// TIA Portal project "Zanzeta_L01_190722" (V16)

(* hardware
DEVICE "S7-1200 station_1"  S7-1200 Station
   slot 0: "Rack_0"  S7-1200 Rack  Rack  V1.0
   slot 1: "PLC_1"  CPU 1215C DC/DC/Rly  6ES7 215-1HG40-0XB0  V4.4
*)

// ===== PLC "PLC_1"  CPU 1215C DC/DC/Rly =====

VAR_GLOBAL   // PLC tag table "Default tag table"
   "Tag_1" AT %MD100 : DInt;
   "Tag_2" AT %MW101 : Int;
   "Tag_3" AT %MD102 : Real;
   "Tag_4" AT %I0.0 : Bool;
   "Tag_5" AT %M0.0 : Bool;
   "Tag_6" AT %MW104 : Int;
   "Tag_7" AT %I0.7 : Bool;
   "Tag_8" AT %Q0.1 : Bool;
END_VAR

// folder: LBC

TYPE "LBC_typeDiagnostics"
TITLE = LBC_typeDiagnostic
// Module related diagnostic information
   STRUCT
      status : Word;   // 16#0000-16#7FFF: Status of the FB 16#8000-16#FFFF: Error identification
      subfunctionStatus : Word;   // Status or return value of called FB's, FCs, system blocks or other status information
      stateNumber : DInt;   // State in the state machine of the block where the error occurred
   END_STRUCT;
END_TYPE

TYPE "LBC_typeInterfaceCommands"
TITLE = LBC_typeInterfaceCommands
// Module related commands from external systems
   STRUCT
      refreshConfiguration : Bool;   // TRUE: Copy global configuration parameters into module interface for external systems
      editConfiguration : Bool;   // TRUE: Edit mode for configuration parameters in control system is active - copying into module interface is stopped
      saveConfiguration : Bool;   // TRUE: Save configuration parameters from module interface into to global configuration parameters after change
      acknowledge : Bool;   // TRUE: Module error acknowledge / reset of errors in function block
   END_STRUCT;
END_TYPE

// folder: LBC/AnalogSignals/Scale

TYPE "LBC_typeAnalogScaleInterface"
TITLE = LBC_typeAnalogScaleInterface
// Module interface for external systems
   STRUCT
      commands : "LBC_typeInterfaceCommands";
      configuration : "LBC_typeAnalogScaleConfiguration";
      monitoring : "LBC_typeAnalogScaleValues";
      diagnostics : "LBC_typeDiagnostics";
   END_STRUCT;
END_TYPE

TYPE "LBC_typeAnalogScaleValues"
TITLE = LBC_typeAnalogScaleValues
// Module related monitoring information
   STRUCT
      enable : Bool;   // TRUE: Enable functionality of FB
      simulation : Bool;   // TRUE: Enable simulation input of input value
      inputValue : LReal;   // Value to be converted
      outputValue : LReal;   // Processed and scaled value
      minValueReached : Bool;   // Minimum configured process value reached. Value is limited to the minimum configured value.
      maxValueReached : Bool;   // Maximum configured process value reached. Value is limited to the maximum configured value.
      error : Bool;   // TRUE: An error occurred while processing the FB
   END_STRUCT;
END_TYPE

TYPE "LBC_typeAnalogScaleConfiguration"
TITLE = LBC_typeAnalogScaleConfiguration
// Module related configuration parameters
   STRUCT
      referenceDesignator : String[20] := 'AnalogScale';   // Device name or device ID
      physicalUnitInput : String[10] := 'unit';   // Physical unit (like [°C], [kWh], etc.) for the input value
      physicalUnitOutput : String[10] := 'unit';   // Physical unit (like [°C], [kWh], etc.) for the output value
      default : LReal := 0.0;   // Default OUTPUT value to be returned if function block is not enabled or quality is bad
      inputValueMax : LReal := 100.0;   // Maximum limit of the process value
      inputValueMin : LReal := -100.0;   // Minimum limit of the process value
      scaleInputUppPoint : LReal := 100.0;   // Upper point for the process value
      scaleInputLowPoint : LReal := -100.0;   // Lower point for the process value
      scaleOutputUppPoint : LReal := 200.0;   // Upper point for the analog process output
      scaleOutputLowPoint : LReal := -200.0;   // Lower point for the analog process output
      disableAlarms : Bool;   // TRUE: Disable the alarms of the block
   END_STRUCT;
END_TYPE

// folder: (top level)

DATA_BLOCK "CMD_PROS_DB"   // DB1
{ S7_Optimized_Access := 'TRUE' }
VERSION : 0.1
// stored: InstanceOfName CMD_PROS
"CMD_PROS"
BEGIN
END_DATA_BLOCK

DATA_BLOCK "TemplateStateMachine_DB"   // DB5
{ S7_Optimized_Access := 'TRUE' }
VERSION : 0.1
// stored: InstanceOfName TemplateStateMachine
"TemplateStateMachine"
BEGIN
END_DATA_BLOCK

// folder: DB

DATA_BLOCK "GlobalDB"   // DB2
{ S7_Optimized_Access := 'TRUE' }
VERSION : 0.1
   VAR RETAIN
      outScale_1 : Real;
      outScale_2 : DInt;
   END_VAR
   VAR
      spMin_1 : Int := 0;
      spMax1 : Int := 27468;
      spMin_2 : Real := 0.0;
      spMax_2 : Real := 20.0;
   END_VAR
   VAR RETAIN
      State_Value : Byte := 2;
   END_VAR
BEGIN
END_DATA_BLOCK

DATA_BLOCK "DB1_IO"   // DB3
{ S7_Optimized_Access := 'TRUE' }
VERSION : 0.1
   VAR
      DBX : Array[0..16] of Bool;
      DBY : Array[0..16] of Bool;
   END_VAR
   VAR RETAIN
      AX1 : DInt;
      AY1 : DInt;
   END_VAR
BEGIN
   DBX[0] := true;
   DBX[1] := true;
END_DATA_BLOCK

DATA_BLOCK "Alarm_DB"   // DB4
{ S7_Optimized_Access := 'TRUE' }
VERSION : 0.1
   VAR
      Alarm_Bool : Array[0..15] of Bool;
   END_VAR
BEGIN
END_DATA_BLOCK

// folder: (top level)

FUNCTION_BLOCK "CMD_PROS"   // FB1, LAD
{ S7_Optimized_Access := 'TRUE' }
VERSION : 0.1
BEGIN
END_FUNCTION_BLOCK

FUNCTION_BLOCK "TemplateStateMachine"   // FB2, LAD
{ S7_Optimized_Access := 'TRUE' }
VERSION : 0.1
   VAR_INPUT
      Actual_Step : Byte;
      Desire_Step : Byte;
      Number_Step : Byte;
      Action_Condirion : Byte;
      Safety_Condition : Byte;
      Interlock : Bool;
      Transition_Condition : Bool;
      Exceptional_Transition : Bool;
      Value : Byte;
   END_VAR
   VAR_OUTPUT
      Actual_Step_1 : Byte;
      Action1 : Bool;
      Action2 : Bool;
      Action3 : Byte;
   END_VAR
   VAR_TEMP   // added for the SCL form of the ladder/FBD networks
      _w1 : Bool;
   END_VAR
BEGIN

REGION Network 1
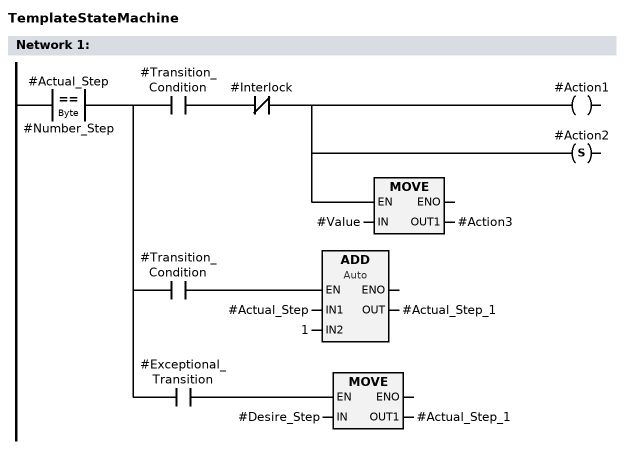
   RUNG wire#powerrail
      { S7_Templates := "SrcType := Byte" } EQ_Contact(in1 := #Actual_Step, in2 := #Number_Step)
      wire#w1
      Contact( #Transition_Condition )
      I_Contact( #Interlock )
      wire#w2
      Coil( #Action1 )
   END_RUNG
   RUNG wire#w2
      S_Coil( #Action2 )
   END_RUNG
   RUNG wire#w2
      Move(in := #Value, out1 => #Action3)
   END_RUNG
   RUNG wire#w1
      Contact( #Transition_Condition )
      Add(in1 := #Actual_Step, in2 := 1, out => #Actual_Step_1)
   END_RUNG
   RUNG wire#w1
      Contact( #Exceptional_Transition )
      Move(in := #Desire_Step, out1 => #Actual_Step_1)
   END_RUNG
   // the same network as SCL:
   #_w1 := #Actual_Step = #Number_Step;
   #Action1 := #_w1 AND #Transition_Condition AND NOT #Interlock;
   IF #Action1 THEN
       #Action2 := TRUE;
       #Action3 := #Value;
   END_IF;
   IF #_w1 AND #Transition_Condition THEN #Actual_Step_1 := #Actual_Step + 1; END_IF;
   IF #_w1 AND #Exceptional_Transition THEN #Actual_Step_1 := #Desire_Step; END_IF;
END_REGION
END_FUNCTION_BLOCK

FUNCTION_BLOCK "LBC_AnalogScale"   // FB22004, SCL
TITLE = LBC_AnalogScale
{ S7_Optimized_Access := 'TRUE' }
AUTHOR : Siemens_Digital_Industry
FAMILY : LBC
NAME : LBC_AnalogScale
// The function is used for processing (scaling) an analog process value to another process value of a different range.  
// Converts it from one to another meaningful unit, e.g. $[rpm]$ to $[m/s]$, $[°C]$ to $[°F]$.
   VAR_INPUT
      enable : Bool;   // TRUE: Enable functionality of FB
      inputValue : LReal;   // Value to be converted
      simulation : Bool;   // TRUE: Enable simulation (input value)
      simulatedInputValue : LReal;   // Simulated input value
   END_VAR
   VAR_OUTPUT
      error : Bool;   // FALSE: No error TRUE: An error occurred during the execution of the FB
      status : Word := 16#7000;   // 16#0000-16#7FFF: Status of the FB 16#8000-16#FFFF: Error identification (see following Table)
      outputValue : LReal;   // Processed and scaled value
      maxValueReached : Bool;   // Maximum configured process value reached. Value is limited to the maximum configured value.
      minValueReached : Bool;   // Minimum configured process value reached. Value is limited to the minimum configured value.
   END_VAR
   VAR_IN_OUT
      configuration : "LBC_typeAnalogScaleConfiguration";
      moduleInterface : "LBC_typeAnalogScaleInterface";
   END_VAR
   VAR
      statProcessValues : "LBC_typeAnalogScaleValues";
      statDiagnostics : "LBC_typeDiagnostics";
      statReferenceDesignator : String[20];   // Device name or device ID
      statLimitationMessage : String[40];   // String to collect information for alarm message of value limitation
      statDisableAlarms : Bool;   // TRUE: Disable the alarms of the block
      statEnablePrevious : Bool;   // Previous value of 'enable' input
   END_VAR
   VAR CONSTANT
      STATUS_NO_ERROR_OCCURRED : Word := 16#0000;   // Status: No error occurred during execution
      STATUS_NO_CALL : Word := 16#7000;   // Status: Function block is not enabled
      STATUS_ENABLED : Word := 16#7002;   // Status: Function block is enabled
      ERR_RANGE_PARAMETRIZATION : Word := 16#8201;   // Error: Configuration range of parameters. min >= max
      ERR_SCALE_ANALOG_POINTS : Word := 16#8202;   // Error: Configuration of analog input points. Process Lower >= Upper
   END_VAR
   // statDiagnostics.status := 16#7000;
BEGIN
   REGION BLOCK INFO HEADER
     //===============================================================================
     // Siemens AG / (c)Copyright 2020
     //-------------------------------------------------------------------------------
     // Title:            LBC_AnalogScale
     // Comment/Function: The function is used for processing (scaling) an analog process value to another process value of a different range. 
     //                   Converts it from one to another meaningful unit, e.g. $[rpm]$ to $[m/s]$, $[°C]$ to $[°F]$.
     // Library/Family:   LBC - Library of Basic Control modules
     // Author:           Siemens Digital Industries
     // Tested with:      S7-PLCSIM Advanced 3.0
     // Engineering:      TIA Portal V16
     // Restrictions:     ENO mechanism is not used - forced to true.
     // Requirements:     PLC (S7-1200 / S7-1500)
     //-------------------------------------------------------------------------------
     // Change log table:
     // Version  | Date       | Expert in charge        | Changes applied
     //----------|------------|-------------------------|-----------------------------
     // 01.00.00 | 15.02.2021 | SIMATIC Systems Support | First released version
     //===============================================================================
   END_REGION

   REGION DESCRIPTION
   (/*The analog scale function block converts a process value to another process value of a different range, e.g. $[rpm]$ to $[m/s]$, $[°C]$ to $[°F]$.

   The processing of the function is started by assigning `TRUE` signal to the `enable` input.  
   If the block is enabled (logical `TRUE`) then the output value is scaled according to settings of the block.

   In order to ensure, that scaling works correctly, it is necessary to set the minimum and the maximum values for input and output.

   For further information see the explanation in the picture and math formulas below.

   ## Process chart
   ![LBC_AnalogScale](LBC_AnalogScale.png "LBC_AnalogScale")

   $ dx = x2 - x1 = scaleInputUppPoint - scaleInputLowPoint $  
   $ dy = y2 - y1 = scaleOutputUppPoint - scaleOutputLowPoint $

   ### Math equation
   $ y = \frac{y_2 - y_1}{x_2 - x_1} \cdot (x - x_1) + y_1 $

   $ x = inputValue $  
   $ y = outputValue $  
   $ x_1 = scaleInputLowPoint $  
   $ x_2 = scaleInputUppPoint $  
   $ y_1 = scaleOutputLowPoint $  
   $ y_2 = scaleOutputUppPoint $*/)
   END_REGION DESCRIPTION

   REGION PROCESS INPUT SIGNALS
     // Assign and initialize internal variables
     #statProcessValues.enable := #enable;
     #statProcessValues.simulation := #simulation;

     // Check if simulation is activated
     IF #statProcessValues.simulation THEN
       #statProcessValues.inputValue := #simulatedInputValue;
     ELSE
       #statProcessValues.inputValue := #inputValue;
     END_IF;

     // Reset limit bits
     #statProcessValues.maxValueReached := FALSE;
     #statProcessValues.minValueReached := FALSE;

     // Copy configuration to static for usage in supervision
     #statDisableAlarms := #configuration.disableAlarms;
   END_REGION PROCESS INPUT SIGNALS

   REGION PARAMETER CHECK
     // Check parameter if block is enabled
     IF #statProcessValues.enable THEN
       #statDiagnostics.status := #STATUS_ENABLED;
       // Validation for hardware range limits 
       // Check if parameters for hardware signal limits are within correct values
       IF #configuration.inputValueMin >= #configuration.inputValueMax THEN
         #statProcessValues.outputValue := #configuration.default;
         #statDiagnostics.status := #ERR_RANGE_PARAMETRIZATION;

       ELSIF #configuration.scaleInputLowPoint >= #configuration.scaleInputUppPoint THEN
         #statProcessValues.outputValue := #configuration.default;
         #statDiagnostics.status := #ERR_SCALE_ANALOG_POINTS;
       END_IF;
     END_IF;
   END_REGION PARAMETER CHECK

   REGION ENABLING/DISABLING
     IF #enable AND NOT #statEnablePrevious THEN
       // Copy configuration to static for usage in associated value of supervision
       #statReferenceDesignator := #configuration.referenceDesignator;

       // Initializes moduleInterface configuration with process configuration
       #moduleInterface.configuration := #configuration;
     END_IF;
     #statEnablePrevious := #enable;
   END_REGION ENABLING/DISABLING

   REGION PROCESS LOGIC
     // Use default value and set no call status if block is disabled
     IF NOT #statProcessValues.enable THEN
       #statProcessValues.outputValue := #configuration.default;
       #statDiagnostics.status := #STATUS_NO_CALL;

       // In case of Error return default
     ELSIF #statDiagnostics.status.%X15 THEN
       #statProcessValues.outputValue := #configuration.default;

       // No error - do process
     ELSE
       // Write status message, set no error
       #statDiagnostics.status := #STATUS_NO_ERROR_OCCURRED;

       // Check if process values are within the configured range
       IF #statProcessValues.inputValue < #configuration.inputValueMin THEN
         #statProcessValues.inputValue := #configuration.inputValueMin;
         #statProcessValues.minValueReached := TRUE;
         #statLimitationMessage := CONCAT(IN1 := LREAL_TO_STRING(#statProcessValues.inputValue), IN2 := #configuration.physicalUnitInput, IN3 := ' <= ', IN4 := LREAL_TO_STRING(#configuration.inputValueMin), IN5 := #configuration.physicalUnitOutput);

       ELSIF #statProcessValues.inputValue > #configuration.inputValueMax THEN
         #statProcessValues.inputValue := #configuration.inputValueMax;
         #statProcessValues.maxValueReached := TRUE;
         #statLimitationMessage := CONCAT(IN1 := LREAL_TO_STRING(#statProcessValues.inputValue), IN2 := #configuration.physicalUnitInput, IN3 := ' >= ', IN4 := LREAL_TO_STRING(#configuration.inputValueMax), IN5 := #configuration.physicalUnitOutput);

       ELSE // Clear alarm message string
         #statLimitationMessage := '';
       END_IF;

       // Scaling the process input
       #statProcessValues.outputValue := (((#statProcessValues.inputValue - #configuration.scaleInputLowPoint) / (#configuration.scaleInputUppPoint - #configuration.scaleInputLowPoint))
       * (#configuration.scaleOutputUppPoint - #configuration.scaleOutputLowPoint) + #configuration.scaleOutputLowPoint);

     END_IF;
   END_REGION PROCESS LOGIC

   REGION CONFIGURATION HANDLING
     // Refresh module interface configuration with process configuration
     IF #moduleInterface.commands.refreshConfiguration AND NOT #moduleInterface.commands.editConfiguration THEN
       #moduleInterface.configuration := #configuration;
     END_IF;
     #moduleInterface.commands.refreshConfiguration := FALSE;

     // Save module interface configuration to process configuration
     IF #moduleInterface.commands.saveConfiguration AND #moduleInterface.commands.editConfiguration THEN
       #configuration := #moduleInterface.configuration;
       #statReferenceDesignator := #configuration.referenceDesignator;
       #moduleInterface.commands.saveConfiguration := FALSE;
     END_IF;
   END_REGION CONFIGURATION HANDLING

   REGION PROCESS OUTPUT SIGNALS
     REGION Write Process data to module interface
       #statProcessValues.error := #statDiagnostics.status.%X15;
       #moduleInterface.monitoring := #statProcessValues;
       #moduleInterface.diagnostics := #statDiagnostics;
     END_REGION Write Process data to module interface

     REGION Write work data to interface and outputs    
       // Write application specific static values to outputs
       #outputValue := #statProcessValues.outputValue;
       #minValueReached := #statProcessValues.minValueReached;
       #maxValueReached := #statProcessValues.maxValueReached;

       // Function status
       #error := #statDiagnostics.status.%X15;
       #status := #statDiagnostics.status;
       // ENO mechanism disabled, ENO - forced to true
       ENO := TRUE;
     END_REGION Write static values to outputs
   END_REGION
END_FUNCTION_BLOCK

FUNCTION "Scalling" : Void   // FC1, LAD
{ S7_Optimized_Access := 'TRUE' }
VERSION : 0.1
   VAR_INPUT
      inMin1 : DInt;
      inMax1 : DInt;
      inMin2 : Real;
      inMax2 : Real;
      inValue : DInt;
   END_VAR
   VAR_OUTPUT
      outReal : LReal;
   END_VAR
   VAR_TEMP
      tempOutNorm1 : LReal;
   END_VAR
BEGIN

REGION Network 1
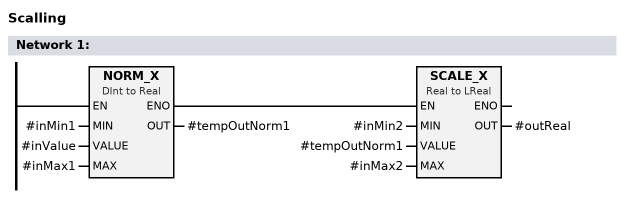
   RUNG wire#powerrail
      { S7_Templates := "[SrcType := DInt, DestType := Real]" } Normalize(min := #inMin1, value := #inValue, max := #inMax1, out => #tempOutNorm1)
      { S7_Templates := "[SrcType := Real, DestType := LReal]" } Scale(min := #inMin2, value := #tempOutNorm1, max := #inMax2, out => #outReal)
   END_RUNG
   // the same network as SCL:
   #tempOutNorm1 := NORM_X(MIN := #inMin1, VALUE := #inValue, MAX := #inMax1);
   #outReal := SCALE_X(MIN := #inMin2, VALUE := #tempOutNorm1, MAX := #inMax2);
END_REGION
END_FUNCTION

FUNCTION "RunMainMotor" : Void   // FC2, LAD
{ S7_Optimized_Access := 'TRUE' }
VERSION : 0.1
BEGIN

REGION Network 1
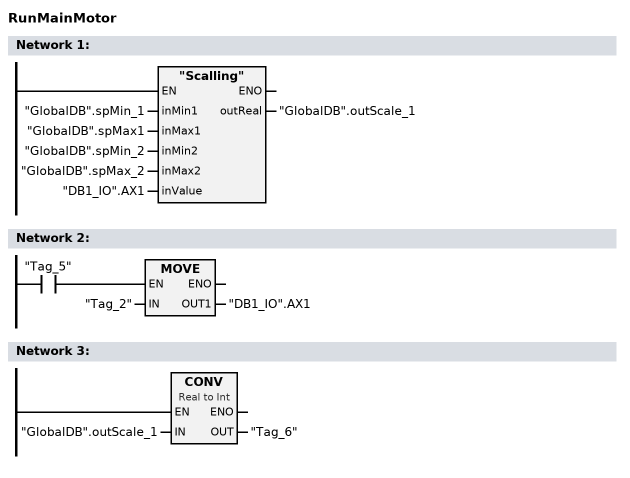
   RUNG wire#powerrail
      "Scalling"(inMin1 := "GlobalDB".spMin_1, inMax1 := "GlobalDB".spMax1, inMin2 := "GlobalDB".spMin_2, inMax2 := "GlobalDB".spMax_2, inValue := "DB1_IO".AX1, outReal => "GlobalDB".outScale_1)
   END_RUNG
   // the same network as SCL:
   "Scalling"(inMin1 := "GlobalDB".spMin_1,
              inMax1 := "GlobalDB".spMax1,
              inMin2 := "GlobalDB".spMin_2,
              inMax2 := "GlobalDB".spMax_2,
              inValue := "DB1_IO".AX1,
              outReal => "GlobalDB".outScale_1);
END_REGION

REGION Network 2
   RUNG wire#powerrail
      Contact( "Tag_5" )
      Move(in := "Tag_2", out1 => "DB1_IO".AX1)
   END_RUNG
   // the same network as SCL:
   IF "Tag_5" THEN "DB1_IO".AX1 := "Tag_2"; END_IF;
END_REGION

REGION Network 3
   RUNG wire#powerrail
      { S7_Templates := "[SrcType := Real, DestType := Int]" } Convert(in := "GlobalDB".outScale_1, out => "Tag_6")
   END_RUNG
   // the same network as SCL:
   "Tag_6" := REAL_TO_INT("GlobalDB".outScale_1);
END_REGION
END_FUNCTION

FUNCTION "IO_ASSIGMENT" : Void   // FC3, LAD
{ S7_Optimized_Access := 'TRUE' }
VERSION : 0.1
BEGIN

REGION Network 1 (SCL)
   REGION io
       // Statement section REGION

   END_REGION
END_REGION
END_FUNCTION

FUNCTION "IO_ASSIGMENT2" : Void   // FC4, SCL
{ S7_Optimized_Access := 'TRUE' }
VERSION : 0.1
BEGIN
END_FUNCTION

FUNCTION "Running_Manual" : Void   // FC5, LAD
{ S7_Optimized_Access := 'TRUE' }
VERSION : 0.1
BEGIN

REGION Network 1
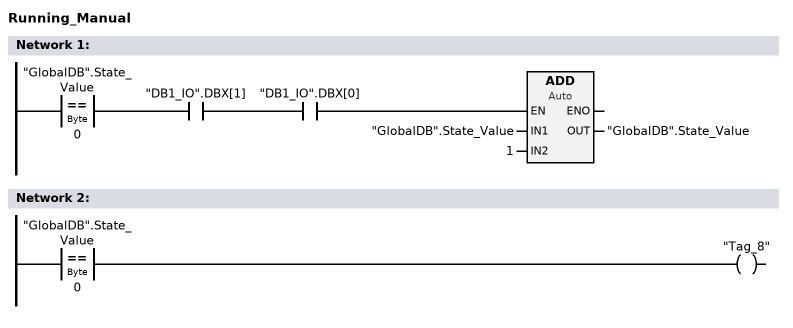
   RUNG wire#powerrail
      { S7_Templates := "SrcType := Byte" } EQ_Contact(in1 := "GlobalDB".State_Value, in2 := 0)
      Contact( "DB1_IO".DBX[1] )
      Contact( "DB1_IO".DBX[0] )
      Add(in1 := "GlobalDB".State_Value, in2 := 1, out => "GlobalDB".State_Value)
   END_RUNG
   // the same network as SCL:
   IF ("GlobalDB".State_Value = 0) AND "DB1_IO".DBX[1] AND "DB1_IO".DBX[0] THEN
       "GlobalDB".State_Value := "GlobalDB".State_Value + 1;
   END_IF;
END_REGION

REGION Network 2
   RUNG wire#powerrail
      { S7_Templates := "SrcType := Byte" } EQ_Contact(in1 := "GlobalDB".State_Value, in2 := 0)
      Coil( "Tag_8" )
   END_RUNG
   // the same network as SCL:
   "Tag_8" := "GlobalDB".State_Value = 0;
END_REGION
END_FUNCTION

ORGANIZATION_BLOCK "Main"   // OB1, LAD, ProgramCycle
TITLE = "Main Program Sweep (Cycle)"
{ S7_Optimized_Access := 'TRUE' }
VERSION : 0.1
   VAR_INPUT
      Initial_Call : Bool;   // Initial call of this OB
      Remanence : Bool;   // =True, if remanent data are available
   END_VAR
BEGIN

REGION Network 1
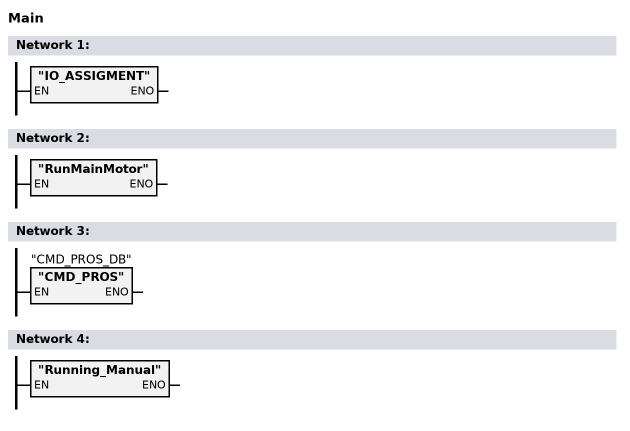
   RUNG wire#powerrail
      "IO_ASSIGMENT"()
   END_RUNG
   // the same network as SCL:
   "IO_ASSIGMENT"();
END_REGION

REGION Network 2
   RUNG wire#powerrail
      "RunMainMotor"()
   END_RUNG
   // the same network as SCL:
   "RunMainMotor"();
END_REGION

REGION Network 3
   RUNG wire#powerrail
      "CMD_PROS_DB"()
   END_RUNG
   // the same network as SCL:
   "CMD_PROS_DB"();   // "CMD_PROS"
END_REGION

REGION Network 4
   RUNG wire#powerrail
      "Running_Manual"()
   END_RUNG
   // the same network as SCL:
   "Running_Manual"();
END_REGION
END_ORGANIZATION_BLOCK

ORGANIZATION_BLOCK "Startup"   // OB100, LAD, Startup
TITLE = "Complete Restart"
{ S7_Optimized_Access := 'TRUE' }
VERSION : 0.1
   VAR_INPUT
      LostRetentive : Bool;   // True if retentive data are lost
      LostRTC : Bool;   // True if date and time are lost
   END_VAR
BEGIN

REGION Network 1
   // Initial Setup
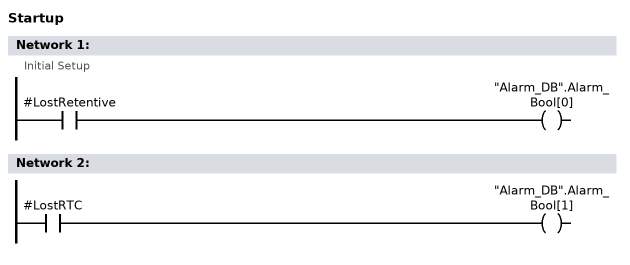
   RUNG wire#powerrail
      Contact( #LostRetentive )
      Coil( "Alarm_DB".Alarm_Bool[0] )
   END_RUNG
   // the same network as SCL:
   "Alarm_DB".Alarm_Bool[0] := #LostRetentive;
END_REGION

REGION Network 2
   RUNG wire#powerrail
      Contact( #LostRTC )
      Coil( "Alarm_DB".Alarm_Bool[1] )
   END_RUNG
   // the same network as SCL:
   "Alarm_DB".Alarm_Bool[1] := #LostRTC;
END_REGION
END_ORGANIZATION_BLOCK

// ===== library types =====

// folder: LGF

FUNCTION "LGF_Description" : Void   // FC10087, SCL
TITLE = LGF_Description
{ S7_Optimized_Access := 'TRUE' }
// Block for the Libray description
BEGIN

   REGION INFO
     (/*title: Library of General Functions (LGF) for SIMATIC S7-1200 / S7-1500
   subTitle: STEP 7 Basic/Professional (TIA PORTAL)
   fileName: LGF
   siosId: 109479728
   link: https://support.industry.siemens.com/cs/ww/en/view/109479728
   version: V5.1.0
   date: 11/2021
   classification:   
   # " " "Frei verwendbar" "Unrestricted" "Intern" "Restricted" "Vertraulich" "Confidential" "Streng vertraulich" "Strictly Confidential"
   title: Library of General Functions (LGF) für SIMATIC S7-1200 / S7-1500
   subTitle: STEP 7 Basic/Professional (TIA PORTAL)
   fileName: LGF
   siosId: 109479728
   link: https://support.industry.siemens.com/cs/ww/de/view/109479728
   version: V5.1.0
   date: 11/2021
   classification:   
   # " " "Frei verwendbar" "Unrestricted" "Intern" "Restricted" "Vertraulich" "Confidential" "Streng vertraulich" "Strictly Confidential"*/)
   END_REGION INFO

   REGION PREAMBLE
     (/*# Library overview

   ## General information

   TIA Portal has an extensive number of "ready-to-use" instructions (mathematical functions, times, counters, etc.). In addition, there are other useful basic functions.

   These functions are provided in the form of a library and they can be used freely. The finished functions are freely customizable and can therefore be used universally.

   The library described here is versioned and it will be continuously extended. For information on versioning, see Chapter "Versioning".

   ## Hardware and software requirements

   #### Requirements for this library

   In order to be able to use the functionality of the library described here, the following hardware and software requirements must be met.

   #### Hardware

   All blocks (FB, FC, DB, ...) in the library can be used universally with the following controllers:
   * SIMATIC S7-1200 and SIMATIC S7-1200 F product family  
   (from firmware V4.2)
   * SIMATIC S7-1500 and SIMATIC S7-1500 F product family  
   (from firmware V2.0)
   * Simulation with SIMATIC S7-PLCSIM  
   (from V14)

   #### Software

   * SIMATIC STEP 7 Basic/Professional (TIA PORTAL)

   ---

   NOTE
   :    In general, it is possible to open a library with STEP 7 Basic, although STEP 7 Professional elements (e.g. SIMATIC S7-1500 controller) are included. In this case you will be informed with a message when opening the library.
   :    All elements (types and copy templates) can be used if they are supported by the hardware installed in the TIA Portal.
   :    If you try to copy elements with STEP 7 Basic from the library that are not supported (e.g. SIMATIC S7-1500 controller), an error message is displayed.
   # Bibliotheksübersicht

   ## Allgemein

   TIA Portal hat eine umfangreiche Anzahl an "ready-to-use" Anweisungen (Mathematische Funktionen, Zeiten, Zähler, usw.). Darüber hinaus gibt es noch weitere nützliche Basisfunktionen.

   Diese Funktionen werden in Form einer Bibliothek zur Verfügung gestellt und können frei verwendet werden. Die fertigen Funktionen sind frei anpassbar und können somit universell eingesetzt werden.

   Die hier beschriebene Bibliothek ist versioniert und wird kontinuierlich erweitert. Informationen zur Versionierung finden Sie im Anhang Kapitel "Versionierung".

   ## Hard- und Softwarevoraussetzungen

   #### Voraussetzungen für diese Bibliothek

   Um die Funktionalität der hier beschriebenen Bibliothek nutzen zu können, sind nachfolgend genannte Hard- und Softwarevoraussetzungen einzuhalten.

   #### Hardware

   Alle Bausteine (FB, FC, DB, …) in der Bibliothek sind universal mit folgenden Steuerungen einsetzbar:
   * SIMATIC S7-1200 und SIMATIC S7-1200 F Produktfamilie  
   (ab Firmware V4.2)
   * SIMATIC S7-1500 und SIMATIC S7-1500 F Produktfamilie  
   (ab Firmware V2.0)
   * Simulation mit SIMATIC S7-PLCSIM  
   (ab V14)

   #### Software

   * SIMATIC STEP 7 Basic/Professional (TIA PORTAL)

   ---

   Hinweis
   :    Es ist generell möglich eine Bibliothek mit STEP 7 Basic zu öffnen, obwohl STEP 7 Professional Elemente (z.B. SIMATIC S7-1500 Steuerung) enthalten sind. In diesem Fall werden Sie mit einer Meldung beim Öffnen der Bibliothek informiert.   
   :    Es können alle Elemente (Typen und Kopiervorlagen) verwendet werden, wenn sie von der installierten Hardware im TIA Portal unterstützt werden.
   :    Falls Sie versuchen Elemente mit STEP 7 Basic aus der Bibliothek zu kopieren, die nicht unterstützt werden (z.B. SIMATIC S7-1500 Steuerung), wird eine Fehlermeldung angezeigt.*/)

     (/*# Working with the library

   ## General information

   All blocks in the "LGF" library can be used freely in conjunction with SIMATIC S7-1200 and SIMATIC S7-1500 controllers.

   Most of the blocks are stored as types in the library. This means that the blocks are versioned and can thus use all advantages.
   * Central update function for library elements
   * Versioning of library elements

   ---

   Note
   :    Information on the general handling of libraries is provided in the Guideline for Library Handling  
   https://support.industry.siemens.com/cs/ww/en/view/109747503  
   :    and in the Programming Guideline for S7-1200/1500 in the chapter "Libraries".  
   https://support.industry.siemens.com/cs/ww/en/view/81318674

   ---

   Note
   :    All blocks in the LGF were created in accordance with the Programming Style Guide.  
   https://support.industry.siemens.com/cs/ww/en/view/81318674

   ---

   For more information on libraries, visit the TIA Portal:
   * Libraries in the TIA Portal  
     https://support.industry.siemens.com/cs/ww/en/view/109738702

   * How do you open libraries in STEP 7 (TIA Portal)?  
   https://support.industry.siemens.com/cs/ww/en/view/37364723

   * Automate in less than 10 minutes TIA Portal: Time Savers – Global libraries  
     https://support.industry.siemens.com/cs/ww/en/view/78529894

   * Which elements from STEP 7 (TIA Portal) can be stored in a library as a type or as a copy template?  
     https://support.industry.siemens.com/cs/ww/en/view/109476862

   * How can you automatically open a global library when starting TIA Portal V13 or higher and use it e.g. as a corporate library?  
     https://support.industry.siemens.com/cs/ww/en/view/100451450

   * Library with PLC data types for IO module / technology modules and PROFIdrive drives (LPD)  
     https://support.industry.siemens.com/cs/ww/en/view/109482396

   ------

   ## Simulation capability with SIMATIC S7-PLCSIM Advanced

   Simulation with SIMATIC S7-PLCSIM Advanced is already activated in the
   properties of the LGF blocks.

   ![Block properties](LIB_Simulation_01.PNG)

   After translation with SIMATIC S7-PLCSIM Advanced, proceed as follows so that
   the blocks can be simulated.

   1. Open the properties of your project and activate the option "Support simulation during block compilation" in the "Protection" tab.

   ![Project properties](LIB_Simulation_00.PNG)

   ---

   Note
   :    Blocks with activated simulation capability take up more memory space in the PLC.

   ------

   ## User-defined documentation (user help)

   In order to explain the principle of operation and use of the blocks to users of the LGF library, user-defined documentation has been created for each block.  
   The user-defined documentation per block is available in German and English as a PDF file. The PDF files are stored in the following directories of the LGF library.

   * German: `"UserFiles\UserDocumentation\en-DE\Library Types"`
   * English: `"UserFiles\UserDocumentation\en-US\Library Types"`

   The user-defined documentation for a block can be called up in the Task Card "Library" and in the library view with the key combination `<Shift+F1>`.  
   The respective PDF is always opened with the standard program defined in Microsoft Windows.

   So that the user-defined documentation of the blocks can also be called up in the project navigation, you must copy the directories with the PDF files into the project directory `UserFiles`.

   ---

   Note
   :    For user-defined documentation, you require SIMATIC STEP 7 Basic / Professional V15.1 Update 1.

   #### Central directory for user-defined documentation

   Alternatively, you can store the user-defined documentation in a central directory for all projects. To define a central storage location for user help, proceed as follows:

   1. In the "Options" menu, select the "Settings" command.
   2. Open the area "General > General".
   3. Navigate to the "User documentation" section.
   4. Activate the checkbox "Display call log for user-defined documentation" to display a log of the call-up of the user-defined documentation in the Inspector window.
   5. Activate the "Search for user-defined documentation in a central directory" checkbox to store user-defined documentation in a central directory for projects.
   6. In the "Central directory for user-defined documentation" field, specify the path where you want to store cross-project documentation.

   ------

   ![Central directory for user defined documentation](LIB_UserDokumentation.PNG)

   ---

   Note
   :    Do not change the names of the PDF, because the file name must precisely match the name of the object in the TIA Portal.

   ---

   Note
   :    Further information on the user-defined documentation can be found in the system manual "SIMATIC STEP 7 Basic/Professional V15.1 and SIMATIC WinCC V15.1":  
   https://support.industry.siemens.com/cs/ww/en/view/109755202/114872699275
   # Arbeiten mit der Bibliothek

   ## Allgemein

   Alle Bausteine in der Bibliothek "LGF" sind frei verwendbar in Verbindung mit SIMATIC S7-1200 und SIMATIC S7-1500 Steuerungen.

   Der Großteil der Bausteine ist als Typ in der Bibliothek abgelegt. Somit sind die Bausteine versioniert und können somit alle Vorteile nutzen.
   * Zentrale Updatefunktion von Bibliothekselementen
   * Versionierung von Bibliothekselementen

   ---

   Hinweis
   :    Informationen zum generellen Umgang mit Bibliotheken finden Sie im Leitfaden zur Bibliothekshandhabung  
   https://support.industry.siemens.com/cs/ww/de/view/109747503  
   :    und im Programmierleitfaden für S7-1200/1500 im Kapitel "Bibliotheken"  
   https://support.industry.siemens.com/cs/ww/de/view/81318674

   ---

   Hinweis
   :    Alle Bausteine in der LGF wurden nach dem Programmierstyleguide erstellt. https://support.industry.siemens.com/cs/ww/de/view/81318674

   ---

   Weitere Informationen zu Bibliotheken im TIA Portal:
   * Themenseite Bibliotheken  
     https://support.industry.siemens.com/cs/ww/de/view/109738702

   * Wie öffnen Sie Bibliotheken in STEP 7 (TIA Portal)?  
     https://support.industry.siemens.com/cs/ww/de/view/37364723

   * Automatisieren in weniger als 10 Minuten TIA Portal: Time Savers – Globale Bibliotheken  
     https://support.industry.siemens.com/cs/ww/de/view/78529894

   * Welche Elemente aus STEP 7 (TIA Portal) können in einer Bibliothek als Typ oder als Kopiervorlage abgelegt werden?  
     https://support.industry.siemens.com/cs/ww/de/view/109476862

   * Wie können Sie beim Starten von TIA Portal ab V13 eine globale Bibliothek automatisch öffnen und z.B. als Unternehmensbibliothek verwenden?  
     https://support.industry.siemens.com/cs/ww/de/view/100451450

   * Bibliothek mit PLC-Datentypen für Peripherie- / Technologie-Module und PROFIdrive Antriebe (LPD)  
     https://support.industry.siemens.com/cs/ww/de/view/109482396

   ------

   ## Simulierbarkeit mit SIMATIC S7-PLCSIM Advanced

   In den Eigenschaften der LGF Bausteine ist die Simulation mit SIMATIC S7-PLCSIM Advanced bereits aktiviert.

   ![Block properties](LIB_Simulation_01.PNG)

   Damit die Bausteine nach dem Übersetzen mit SIMATIC S7-PLCSIM Advanced
   simuliert werden können, gehen Sie folgendermaßen vor:

   1. Öffnen Sie die Eigenschaften Ihres Projekts und aktivieren Sie im Register "Schutz" die Option "Beim Übersetzen von Bausteinen Simulierbarkeit unterstützen" ("Support simulation during block compilation").

   ![Project properties](LIB_Simulation_00.PNG)

   ---

   Hinweis
   :    Bausteine mit aktivierter Simulierbarkeit belegen mehr Speicherplatz in der PLC.

   ------

   ## Anwenderdefinierte Dokumentation (Anwenderhilfe)

   Um den Anwendern der Bibliothek LGF die Funktionsweise und die Verwendung der Bausteine zu erläutern, wurde für jeden Baustein eine anwenderdefinierte Dokumentation erstellt.  
   Die anwenderdefinierte Dokumentation pro Bausteine ist in den Sprachen Deutsch und Englisch als PDF-Datei verfügbar. Die PDF-Dateien sind in folgenden Verzeichnissen der Bibliothek LGF gespeichert.

   * Deutsch: `"UserFiles\UserDocumentation\de-DE\Library Types"`
   * Englisch: `"UserFiles\UserDocumentation\en-US\Library Types"`

   Die anwenderdefinierte Dokumentation zu einem Baustein können Sie in der Task Card "Bibliothek" und in der Bibliotheksansicht mit der Tastenkombination `<Shift+F1>` aufrufen.  
   Die jeweilige PDF wird immer mit dem in Microsoft Windows festgelegten Standardprogramm geöffnet.

   Damit die anwenderdefinierten Dokumentationen der Bausteine auch in der Projektnavigation aufgerufen werden kann, müssen Sie die Verzeichnisse mit den PDF-Dateien in das Projektverzeichnis "UserFiles" kopieren.

   ---

   Hinweis
   :    Für die Anwenderdefinierte Dokumentation benötigen Sie SIMATIC STEP 7 Basic/Professional V15.1 Update 1.

   #### Zentrales Verzeichnis für anwenderdefinierte Dokumentation

   Alternativ können Sie die anwenderdefinierte Dokumentation auch projektüber-greifend in einem zentralen Verzeichnis ablegen. Um einen zentralen Ablageort für Anwenderhilfe festzulegen, gehen Sie folgendermaßen vor:
   1. Wählen Sie im Menü "Extras" ("Options") den Befehl "Einstellungen" ("Settings").
   2. Öffnen Sie den Bereich "Allgemein > Allgemein" ("General > General").
   3. Navigieren Sie zum Abschnitt "Anwenderdokumentation" ("User documentation").
   4. Aktivieren Sie das Optionskästchen "Aufrufprotokoll zu anwenderdefinierter Dokumentation anzeigen" ("Display call log for user-defined documentation"), um im Inspektor Fenster ein Protokoll vom Aufruf der anwenderdefinierten Dokumentation anzuzeigen.
   5. Aktivieren Sie das Optionskästchen "Suche nach anwenderdefinierter Dokumentation in einem zentralen Verzeichnis" ("Search for user-defined documentation in a central directory"), um anwenderdefinierte Dokumentation in einem projektübergreifenden Verzeichnis abzulegen.
   6. Geben Sie im Feld "Zentrales Verzeichnis für anwenderdefinierte Dokumentation" ("Central directory for user-defined documentation") den Pfad an, an dem Sie projektübergreifende Dokumentation speichern.

   ------

   ![Central directory for user defined documentation](LIB_UserDokumentation.PNG)

   ---

   Hinweis
   :    Ändern Sie nicht die Namen der PDF, denn der Dateiname muss exakt dem
   Namen des Objekts im TIA Portal entsprechen.

   ---

   Hinweis
   :    Weitere Informationen zur anwenderdefinierten Dokumentation finden Sie im
   Systemhandbuch "SIMATIC STEP 7 Basic/Professional V15.1 und SIMATIC
   WinCC V15.1" unter:  
   https://support.industry.siemens.com/cs/ww/de/view/109755202/114872699275*/)

     (/*# Explanation of the blocks

   The chapters below describe all blocks of the library, "Library of General Functions".  
   The chapters have the same structure as the library itself.

   All blocks are divided into application areas or categories:
   * Bit logic operations
   * Date and timer operations
   * Counter operations
   * Comparator operations
   * Math operations
   * Data handling
   * Converter operations
   * Signal generators
   * Technology operations
   * Measurement operations

   ![Global Library (LGF)](LGF_ProjectTree.PNG)
   # Erläuterung der Bausteine

   Die folgenden Kapitel beschreiben alle Bausteine der Bibliothek "Library of General Functions".  
   Die Kapitel sind nach der gleichen Struktur aufgebaut wie die Bibliothek selbst.

   Alle Bausteine sind in Anwendungsgebiete bzw. Kategorien eingeteilt:
   * Bit logic operations (Bitoperationen)
   * Date and timer operations (Datum und Zeitoperationen)
   * Counter operations (Zähloperationen)
   * Comparator operations (Vergleichsoperationen)
   * Math operations (mathematische Operationen)
   * Data handling (Datenverarbeitung)
   * Converter operations (Konvertierungsoperationen)
   * Signal generators (Signalgeneratoren)
   * Technology operations (Technologieoperationen)
   * Measurement operations (Messdatenoperationen)

   ![Global Library (LGF)](LGF_ProjectTree.PNG)*/)
   END_REGION PREAMBLE

   REGION APPENDIX
     (/*# Appendix

   ## Service and support

   #### Industry Online Support
   Do you have any questions or need assistance?  
   Siemens Industry Online Support offers round the clock access to our entire service and support know-how and portfolio.  
   The Industry Online Support is the central address for information about our products, solutions and services.  
   Product information, manuals, downloads, FAQs, application examples and videos, all information is accessible with just a few mouse clicks:  
   https://support.industry.siemens.com

   #### Technical Support
   The Technical Support of Siemens Industry provides you fast and competent support regarding all technical queries with numerous tailor-made offers - ranging from basic support to individual support contracts. Please send queries to Technical Support via Web form:  
   https://www.siemens.com/supportrequest

   #### SITRAIN - Digital Industry Academy
   We support you with our globally available training courses for industry with practical experience, innovative learning methods and a concept that's tailored to the customer's specific needs.  
   For more information on our offered trainings and courses, as well as their locations and dates, refer to our web page:  
   https://www.siemens.com/sitrain

   #### Service offer
   Our range of services includes the following:
   * Plant data services
   * Spare parts services
   * Repair services
   * On-site and maintenance services
   * Retrofitting and modernization services
   * Service programs and contract's

   You can find detailed information on our range of services in the service catalog web page:  
   https://support.industry.siemens.com/cs/sc  

   #### Industry Online Support app
   You will receive optimum support wherever you are with the "Siemens Industry Online Support" app. The app is available for iOS and Android:  
   https://support.industry.siemens.com/cs/ww/en/sc/2067

   ## Industry Mall

   ![Siemens Industry Mall](SiemensIndustryMall.png)

   The Siemens Industry Mall is the platform on which the entire Siemens Industry product portfolio is accessible. From the selection of products to the order and the delivery tracking, the Industry Mall enables the complete purchasing processing – directly and independently of time and location:  
   https://mall.industry.siemens.com
   # Anhang

   ## Service und Support

   #### Industry Online Support
   Sie haben Fragen oder brauchen Unterstützung?  
   Über den Industry Online Support greifen Sie rund um die Uhr auf das gesamte Service und Support Know-how sowie auf unsere Dienstleistungen zu.  
   Der Industry Online Support ist die zentrale Adresse für Informationen zu unseren Produkten, Lösungen und Services.  
   Produktinformationen, Handbücher, Downloads, FAQs und Anwendungsbeispiele, alle Informationen sind mit wenigen Mausklicks erreichbar:  
   https://support.industry.siemens.com

   #### Technical Support
   Der Technical Support von Siemens Industry unterstützt Sie schnell und kompetent bei allen technischen Anfragen mit einer Vielzahl maßgeschneiderter Angebote, von der Basisunterstützung bis hin zu individuellen Supportverträgen.  
   Anfragen an den Technical Support stellen Sie per Web-Formular:  
   https://www.siemens.com/supportrequest

   #### SITRAIN – Digital Industry Academy
   Mit unseren weltweit verfügbaren Trainings für unsere Produkte und Lösungen unterstützen wir Sie praxisnah, mit innovativen Lernmethoden und mit einem kundenspezifisch abgestimmten Konzept.  
   Mehr zu den angebotenen Trainings und Kursen sowie deren Standorte und Termine erfahren Sie unter:  
   https://www.siemens.de/sitrain

   #### Serviceangebot
   Unser Serviceangebot umfasst folgendes:
   * Plant Data Services
   * Ersatzteilservices
   * Reparaturservices
   * Vor-Ort und Instandhaltungsservices
   * Retrofit- und Modernisierungsservices
   * Serviceprogramme und Verträge

   Ausführliche Informationen zu unserem Serviceangebot finden Sie im Servicekatalog:  
   https://support.industry.siemens.com/cs/sc

   #### Industry Online Support App
   Mit der App "Siemens Industry Online Support" erhalten Sie auch unterwegs die optimale Unterstützung. Die App ist für iOS und Android verfügbar:  
   https://support.industry.siemens.com/cs/ww/de/sc/2067

   ## Industry Mall

   ![Siemens Industry Mall](SiemensIndustryMall.png)

   Die Siemens Industry Mall ist die Plattform, auf der das gesamte Produktportfolio von Siemens Industry zugänglich ist. Von der Auswahl der Produkte über die Bestellung und die Lieferverfolgung ermöglicht die Industry Mall die komplette Einkaufsabwicklung – direkt und unabhängig von Zeit und Ort:  
   https://mall.industry.siemens.com*/)


     (/*## Links and Literature
   +-----+-----------------------------------------------------------------------+
   | No. |Topic     
   +=====+=======================================================================+
   | \1\ | Siemens Industry Online Support
   |     | https://support.industry.siemens.com 
   +-----+-----------------------------------------------------------------------+
   | \2\ | Link to the entry page of the application example
   |     | https://support.industry.siemens.com/cs/ww/en/view/109479728
   +-----+-----------------------------------------------------------------------+
   | \3\ | Programming Guidelines and Programming Style guide for SIMATIC S7-1200 and S7-1500
   |     | https://support.industry.siemens.com/cs/ww/en/view/81318674
   +-----+-----------------------------------------------------------------------+
   | \4\ | Library with PLC data types (LPD) for STEP 7 (TIA Portal) and SIMATIC S7-1200 / S7-1500
   |     | https://support.industry.siemens.com/cs/ww/en/view/109482396
   +-----+-----------------------------------------------------------------------+
   | \5\ | Guideline on Library Handling in Tia Portal
   |     | https://support.industry.siemens.com/cs/ww/en/view/109747503
   +-----+-----------------------------------------------------------------------+
   | \6\ | Libraries in the TIA Portal
   |     | https://support.industry.siemens.com/cs/ww/en/view/109738702

   ------
   ## Links und Literatur
   +---------+---------+
   | No.     |Topic     
   +=========+=========+
   | \1\     | Siemens Industry Online Support
   |         | https://support.industry.siemens.com 
   +---------+---------+
   | \2\     | Link auf die Beitragsseite des Anwendungsbeispiels
   |         | https://support.industry.siemens.com/cs/ww/de/view/109479728
   +---------+---------+
   | \3\     | Programmierleitfaden und Programmierstyleguide für SIMATIC S7-1200 and S7-1500
   |         | https://support.industry.siemens.com/cs/ww/de/view/81318674
   +---------+---------+
   | \4\     | Bibliothek mit PLC-Datentypen (LPD) für STEP 7 (TIA Portal) und SIMATIC S7-1200 / S7-1500
   |         | https://support.industry.siemens.com/cs/ww/de/view/109482396
   +---------+---------+
   | \5\     | Leitfaden zur Bibliothekshandhabung
   |         | https://support.industry.siemens.com/cs/ww/de/view/109747503
   +---------+---------+
   | \6\     | Themenseite Bibliotheken
   |         | https://support.industry.siemens.com/cs/ww/de/view/109738702

   ------*/)

     (/*## Change documentation

   #### Versioning of the library
   The library and library elements are maintained in accordance with the table below:

   +----+-------------------------------------------+-----------------------------------------+--------------------+
   | P  | 1.                                        | 2.                                      | 3.                 |
   +====+===========================================+=========================================+====================+
   |    | Non-compatible change                     | Compatible change                       | Error correction   |
   +----+-------------------------------------------+-----------------------------------------+--------------------+
   |    | * Reduction of interfaces                 | * Extension of the interfaces           | * Bug fix          |
   |    | * Changing the interfaces                 | * Compatible extension of functionality |                    |
   |    | * Incompatible extension of functionality |                                         |                    |

   #### Versioning example

   Example for changing the version:  

   | Library | FB1 | FB2 | FC1 | FC2 | Comment |
   | --- | --- | --- | --- | --- | --- |
   | 1.0.0 | 1.0.0 | 1.0.0 | 1.0.0 | - | Released | 
   | 1.0.1 | 1.0.1 | 1.0.0 | 1.0.0 | - | Troubleshooting of FB1 | 
   | 1.0.2 | 1.0.1 | 1.0.1 | 1.0.0 | - | Optimization of FB2 | 
   | 1.1.0 | 1.1.0 | 1.0.1 | 1.0.0 | - | Extension to FB1 | 
   | 1.2.0 | 1.2.0 | 1.0.1 | 1.0.0 | - | Extension to FB1 | 
   | 2.0.0 | 2.0.0 | 1.0.1 | 2.0.0 | - | New functionality on FB1 and FC1 | 
   | 2.0.1 | 2.0.0 | 1.0.2 | 2.0.0 | - | Troubleshooting FB2 | 
   | 3.0.0 | 2.0.0 | 1.0.2 | 2.0.0 | 1.0.0 | New function FC2 | 
   | 3.0.1 | 2.0.1 | 1.0.3 | 2.0.1 | 1.0.1 | Upgrade to new TIA Portal version | 
   | 3.0.2 | 2.0.2 | 1.0.4 | 2.0.2 | 1.0.1 | New functions, bug fixes |
   ## Änderungsdokumentation

   #### Versionierung der Bibliothek
   Die Bibliothek und Bibliothekselemente werden gemäß folgender Tabelle gepflegt:

   +----+-----------------------------------------------+---------------------------------------------+-----------------+
   | P  | 1.                                            | 2.                                          | 3.              |
   +====+===============================================+=============================================+=================+
   |    | Nichtkompatible Änderung                      | Kompatible Änderung                         | Fehlerkorrektur |
   +----+-----------------------------------------------+---------------------------------------------+-----------------+
   |    | * Reduzierung der Schnittstellen              | * Erweiterung der Schnittstellen            | * Bugfix        |
   |    | * Ändern der Schnittstellen                   | * Kompatible Erweiterung der Funktionalität |                 |
   |    | * Inkompatible Erweiterung der Funktionalität |                                             |                 |

   #### Versionierungs Beispiel

   Beispiel für das ändern und hochzählen der Versionsnummer:

   |  Library | FB1 | FB2 | FC1 | FC2 | Comment |
   | --- | --- | --- | --- | --- | --- |
   | 1.0.0 | 1.0.0 | 1.0.0 | 1.0.0 | - | freigegeben | 
   | 1.0.1 | 1.0.1 | 1.0.0 | 1.0.0 | - | Fehlerbehebung von FB1 | 
   | 1.0.2 | 1.0.1 | 1.0.1 | 1.0.0 | - | Optimierung von FB2 | 
   | 1.1.0 | 1.1.0 | 1.0.1 | 1.0.0 | - | Erweiterung an FB1 | 
   | 1.2.0 | 1.2.0 | 1.0.1 | 1.0.0 | - | Erweiterung an FB1 | 
   | 2.0.0 | 2.0.0 | 1.0.1 | 2.0.0 | - | neue Funktionalität an FB1 und FC1 | 
   | 2.0.1 | 2.0.0 | 1.0.2 | 2.0.0 | - | Fehlerbehebung FB2 | 
   | 3.0.0 | 2.0.0 | 1.0.2 | 2.0.0 | 1.0.0 | Neue Funktion FC2 | 
   | 3.0.1 | 2.0.1 | 1.0.3 | 2.0.1 | 1.0.1 | Upgrade auf neue TIA Portal Version | 
   | 3.0.2 | 2.0.2 | 1.0.4 | 2.0.2 | 1.0.1 | Neue Funktionen, Fehlerbehebungen |*/)
   END_REGION APPENDIX
END_FUNCTION

// folder: LGF/0 Bit logic operations

FUNCTION "LGF_BitToggle" : DWord   // FC10033, SCL
TITLE = LGF_BitToggle
{ S7_Optimized_Access := 'TRUE' }
AUTHOR : Siemens_SIMATIC_Systems_Support
FAMILY : LGF
NAME : LGF_BitToggle
// Dieser Baustein toggelt (von TRUE nach FALSE und umgekehrt) ein Bit an vorgegebener Stelle in einer Variablen vom Datentyp DWORD.    
// Anstelle von DWord kann auch Word und Byte verwendet werden, indem der übergebene Parameter mit z. B. BYTE_TO_DWORD und das Ergebnis mit DWORD_TO_BYTE konvertiert wird.
// This block toggles (from TRUE to FALSE and vice versa) a bit at a predefined position in a variable of the data type DWORD.  
// Alternatively, Word and Byte can be used instead of DWord by converting the passed parameter with, for example, BYTE_TO_DWORD and the result with DWORD_TO_BYTE
   VAR_INPUT
      value : DWord;   // Tag where the bit has to be toggled / Variable, an der das Bit getoggelt wird.
      bitNo : USInt;   // Bit number to be toggled in the “value” parameter. / Bitnummer, die im Parameter "value" getoggelt werden soll.
   END_VAR
   // Ret_Val : Tag with toggled bit / Variable mit getoggeltem Bit.
   VAR CONSTANT
      TRUE_BOOL_BIT : DWord := 16#0001;   // Just one bit which is true, to shift in Dword for masking / Ein einzelnes Bit mit Wert := TRUE zum schieben im Dword und zur Maskierung
      MAX_NO_OF_BITS : USInt := 32;   // Maximum bits in a DWord = 32 / Maximalanzahl an Bits in einem Dword = 32
   END_VAR
BEGIN
   REGION BLOCK INFO HEADER
     //===============================================================================
     // SIEMENS AG / (c)Copyright 2019
     //-------------------------------------------------------------------------------
     // Title:            LGF_BitToggle
     // Comment/Function: Toggle bit in elementary datatype - DWord
     //                   can be used for Word and Byte as well, by convert
     //                   the passed paramter and the result using for e.g. Dword_to_Byte
     // Library/Family:   LGF (Library General Functions)
     // Author:           Siemens Digital Industry
     // Tested with:      CPU1212C DC/DC/DC FW:V4.2
     // Engineering:      TIA Portal V15.1
     // Restrictions:     ENO not in use, set to true, no error handling
     // Requirements:     PLC (S7-1200 / S7-1500)
     //-------------------------------------------------------------------------------
     // Change log table:
     // Version  | Date       | Expert in charge         | Changes applied
     // 01.00.00 | 06.06.2015 | Siemens Industry Support | first release
     // 03.00.00 | 23.04.2020 | Siemens Industry Support | Set version to V3.0.0
     //                         harmonize the version of the whole library
     // 03.00.01 | 19.01.2021 | Simatic Systems Support
     //                         Insert documentation
     //===============================================================================
   END_REGION

   REGION Logic
     // toggle the bit in tag
     // shift one true bit into given position
     // concatenate value then with XOR resets the bit on the given position
     #LGF_BitToggle := #value XOR SHL(IN := #TRUE_BOOL_BIT, N := (#bitNo MOD #MAX_NO_OF_BITS));

     // no error handling needed
     ENO := TRUE;
   END_REGION
END_FUNCTION

FUNCTION "LGF_BitTest" : Bool   // FC10076, SCL
TITLE = LGF_BitTest
{ S7_Optimized_Access := 'TRUE' }
AUTHOR : Siemens_SIMATIC_Systems_Support
FAMILY : LGF
NAME : LGF_BitTest
// Dieser Baustein prüft ein Bit an vorgegebener Stelle in einer Variablen vom Daten-typ DWORD auf TRUE oder FALSE.  
// Anstelle von DWord kann auch Word und Byte verwendet werden, indem der übergebene Parameter mit z. B. BYTE_TO_DWORD und das Ergebnis mit DWORD_TO_BYTE konvertiert wird.
// This block checks whether a bit is TRUE or FALSE at a given position in a variable of the data type DWORD.  
// Alternatively, Word and Byte can be used instead of DWord by converting the passed parameter with, for example, BYTE_TO_DWORD and the result with DWORD_TO_BYTE.
   VAR_INPUT
      value : DWord;   // Tag where the bit has to be tested / Variable, an der das Bit überprüft wird.
      bitNo : USInt;   // bit number to test in "value" parameter / Bitnummer, die im Parameter "value" überprüft werden soll.
   END_VAR
   // Ret_Val : Value of the checked bit. / Wert des überprüften Bits.
   VAR CONSTANT
      BINARY_ZERO : DWord := 16#0000;   // Binary zero to compare shifted result / Binäre null zum vergleich mit dem geschobenen Ergebnis
      TRUE_BOOL_BIT : DWord := 16#0001;   // Just one bit which is true, to shift in Dword for masking / Ein einzelnes Bit mit Wert := TRUE zum schieben im Dword und zur Maskierung
      MAX_NO_OF_BITS : USInt := 32;   // Maximum bits in a DWord = 32 / Maximalanzahl an Bits in einem Dword = 32
   END_VAR
BEGIN
   REGION BLOCK INFO HEADER
     //===============================================================================
     // SIEMENS AG / (c)Copyright 2019
     //-------------------------------------------------------------------------------
     // Title:            LGF_BitTest
     // Comment/Function: Test bit in DWord if it is 1 or 0 respectively
     //                   returning TRUE or FALSE
     //                   can be used for Word and Byte as well, by convert
     //                   the passed paramter and the result using for e.g. Dword_to_Byte
     // Library/Family:   LGF (Library General Functions)
     // Author:           Siemens Digital Industry
     // Tested with:      CPU1212C DC/DC/DC FW:V4.2
     // Engineering:      TIA Portal V15.1
     // Restrictions:     ENO not in use, set to true, no error handling
     // Requirements:     PLC (S7-1200 / S7-1500)
     //-------------------------------------------------------------------------------
     // Change log table:
     // Version  | Date       | Expert in charge         | Changes applied
     // 01.00.00 | 06.06.2015 | Siemens Industry Support | first release
     // 03.00.00 | 23.04.2020 | Siemens Industry Support | Set version to V3.0.0
     //                         harmonize the version of the whole library
     // 03.00.01 | 19.01.2021 | Simatic Systems Support
     //                         Insert documentation
     //===============================================================================
   END_REGION

   REGION Logic
     // test the bit in tag
     // shift one true bit into the selected position
     // compare with input value with "AND" logic and check if different to zero
     // result is true if bit is true, otherwise it is false
     #LGF_BitTest := (#BINARY_ZERO <> (#value AND SHL(IN := #TRUE_BOOL_BIT, N := (#bitNo MOD #MAX_NO_OF_BITS))));

     // no error handling needed
     ENO := TRUE;
   END_REGION
END_FUNCTION

FUNCTION "LGF_BitSet" : DWord   // FC10078, SCL
TITLE = LGF_BitSet
{ S7_Optimized_Access := 'TRUE' }
AUTHOR : Siemens_SIMATIC_Systems_Support
FAMILY : LGF
NAME : LGF_BitSet
// Dieser Baustein setzt ein Bit an vorgegebener Stelle in einer Variable vom Daten-typ DWORD.  
// Anstelle von DWord kann auch Word und Byte verwendet werden, indem der übergebene Parameter mit z. B. BYTE_TO_DWORD und das Ergebnis mit DWORD_TO_BYTE konvertiert wird.
// This block sets a bit at a given position in a variable of the data type DWORD.  
// Alternatively, Word and Byte can be used instead of DWord by converting the passed parameter with, for example, BYTE_TO_DWORD and the result with DWORD_TO_BYTE.
   VAR_INPUT
      value : DWord;   // Tag where the bit has to be set / Variable, an der das Bit gesetzt wird
      bitNo : USInt;   // Bit number to set in "value" parameter / Bitnummer, die im Parameter "value" gesetzt werden soll
   END_VAR
   // Ret_Val : Tag with the set bit / Variable mit gesetztem Bit
   VAR CONSTANT
      TRUE_BOOL_BIT : DWord := 16#0001;   // Just one bit which is true, to shift in Dword for masking / Ein einzelnes Bit mit Wert := TRUE zum schieben im Dword und zur Maskierung
      MAX_NO_OF_BITS : USInt := 32;   // Maximum bits in a DWord = 32 / Maximalanzahl an Bits in einem Dword = 32
   END_VAR
BEGIN
   REGION BLOCK INFO HEADER
     //===============================================================================
     // SIEMENS AG / (c)Copyright 2019
     //-------------------------------------------------------------------------------
     // Title:            LGF_BitSet
     // Comment/Function: Set bit in elementary datatype - DWord
     //                   cam be used for Word and Byte as well, by convert
     //                   the passed paramter and the result using for e.g. Dword_to_Byte
     // Library/Family:   LGF (Library General Functions)
     // Author:           Siemens Digital Industry
     // Tested with:      CPU1212C DC/DC/DC FW:V4.2
     // Engineering:      TIA Portal V15.1
     // Restrictions:     ENO not in use, set to true, no error handling
     // Requirements:     PLC (S7-1200 / S7-1500)
     //-------------------------------------------------------------------------------
     // Change log table:
     // Version  | Date       | Expert in charge         | Changes applied
     // 01.00.00 | 06.06.2015 | Siemens Industry Support | first release
     // 03.00.00 | 23.04.2020 | Siemens Industry Support | Set version to V3.0.0
     //                         harmonize the version of the whole library
     // 03.00.01 | 19.01.2021 | Simatic Systems Support
     //                         Insert documentation
     //===============================================================================
   END_REGION

   REGION Logic
     // set the bit in tag
     // shift one true bit into given position
     // concatenate value then with OR will result in the previous value and the set bit in position
     #LGF_BitSet := #value OR SHL(IN := #TRUE_BOOL_BIT, N := (#bitNo MOD #MAX_NO_OF_BITS));

     // no error handling needed
     ENO := TRUE;
   END_REGION
END_FUNCTION

FUNCTION "LGF_BitReset" : DWord   // FC10080, SCL
TITLE = LGF_BitReset
{ S7_Optimized_Access := 'TRUE' }
AUTHOR : Siemens_SIMATIC_Systems_Support
FAMILY : LGF
NAME : LGF_BitReset
// Dieser Baustein setzt ein Bit an vorgegebener Stelle in einer Variablen vom Daten-typ DWORD zurück.  
// Anstelle von DWord kann auch Word und Byte verwendet werden, indem der übergebene Parameter mit z. B. BYTE_TO_DWORD und das Ergebnis mit DWORD_TO_BYTE konvertiert wird.
// This block resets a bit at a predefined position in a variable of the data type DWORD.  
// Alternatively, Word and Byte can be used instead of DWord by converting the passed parameter with, for example, BYTE_TO_DWORD and the result with DWORD_TO_BYTE.
   VAR_INPUT
      value : DWord;   // Tag where the bit has to be reset / Variable, an der das Bit zurückgesetzt wird.
      bitNo : USInt;   // Bit number to reset in "value" parameter / Bitnummer, die im Parameter "value" zurück gesetzt werden soll
   END_VAR
   // Ret_Val : Tag with reset bit / Variable mit zurückgesetztem Bit.
   VAR CONSTANT
      BINARY_ONES : DWord := 16#FFFFFFFF;   // Binary ones - all bits are true to concatenate shifted result / Binäre EINSEN - alle Bits sind true für die UND Verknüpfung mit dem geschobenen Ergebnis
      TRUE_BOOL_BIT : DWord := 16#0001;   // Just one bit which is true, to shift in Dword for masking / Ein einzelnes Bit mit Wert := TRUE zum schieben im Dword und zur Maskierung
      MAX_NO_OF_BITS : USInt := 32;   // Maximum bits in a DWord = 32
   END_VAR
BEGIN
   REGION BLOCK INFO HEADER
     //===============================================================================
     // SIEMENS AG / (c)Copyright 2019
     //-------------------------------------------------------------------------------
     // Title:            LGF_BitReset
     // Comment/Function: Reset bit in elementary datatype - DWord
     //                   can be used for Word and Byte as well, by convert
     //                   the passed paramter and the result using for e.g. Dword_to_Byte
     // Library/Family:   LGF (Library General Functions)
     // Author:           Siemens Digital Industry
     // Tested with:      CPU1212C DC/DC/DC FW:V4.2
     // Engineering:      TIA Portal V15.1
     // Restrictions:     ENO not in use, set to true, no error handling
     // Requirements:     PLC (S7-1200 / S7-1500)
     //-------------------------------------------------------------------------------
     // Change log table:
     // Version  | Date       | Expert in charge         | Changes applied
     // 01.00.00 | 06.06.2015 | Siemens Industry Support | first release
     // 03.00.00 | 23.04.2020 | Siemens Industry Support | Set version to V3.0.0
     //                         harmonize the version of the whole library
     // 03.00.01 | 19.01.2021 | Simatic Systems Support
     //                         Insert documentation
     //===============================================================================
   END_REGION

   REGION Logic
     // reset the bit in tag
     // shift one true bit into given position
     // concatenate value then with XOR and biary ones
     // using this result with AND and value will result in the previous value and the reseted bit in position
     #LGF_BitReset := #value AND (#BINARY_ONES XOR SHL(IN := #TRUE_BOOL_BIT, N := (#bitNo MOD #MAX_NO_OF_BITS)));

     // no error handling needed
     ENO := TRUE;
   END_REGION
END_FUNCTION